// TIA Portal V19 export
VAR_GLOBAL   // PLC tag table "00_A01_MB1_Tower"
   A01_TowerHorn_SL101 AT %Q121.7 : Bool;   // 370HA1
   A01_TowerLampYellow_SL101 AT %Q121.5 : Bool;   // 370HL1
   A01_TowerLampWhite_SL101 AT %Q121.6 : Bool;   // 370HL2
   MB1_Pb_ResetAlarms AT %I109.0 : Bool;   // 300SH1
   MB1_Loop1_Pb AT %I109.1 : Bool;   // 300SH2
   MB1_Area01_SelMan AT %I109.2 : Bool;   // 300SA1
   MB1_Area01_SelAut AT %I109.3 : Bool;   // 300SA1
   MB1_Area01_PbCycleStart AT %I109.4 : Bool;   // 300SH3
   MB1_Area01_PbCycleStop AT %I109.5 : Bool;   // 300SB1
   MB1_PbJogPlus AT %I109.6 : Bool;   // 301SA1
   MB1_PbJogMInus AT %I109.7 : Bool;   // 301SA1
   MB1_Sel_Material_FWD AT %I110.0 : Bool;   // 301SA2
   MB1_Sel_Material_BWD AT %I110.1 : Bool;   // 301SA2
   MB1_Area01_LpPbReset AT %Q109.7 : Bool;   // 300SH1
   MB1_Lp_Loop1 AT %Q110.0 : Bool;   // 300SH2
   MB1_Area01_LpCycleReady AT %Q110.1 : Bool;   // 300HL1
   MB1_Area01_LpCycleStart AT %Q110.2 : Bool;   // 300SH3
   MB1_LpJog AT %Q110.3 : Bool;   // 301SA1
   MB1_Pb_LIBERO AT %I110.4 : Bool;   // 302 - LIBERO
   MB1_Lp_LIBERO AT %Q110.5 : Bool;   // 302 - LIBERO
   "DecoilersHRot_TowerLamp_SL101-SL102" AT %Q122.0 : Bool;   // 370HL3
END_VAR
